Staubli VAL3: retrieveViews.pgx

public program retrieveViews(viewType& view_, num& idx_)
begin
  switch idx_
    case 0
      view_.path=IMM_IO_PTH
      view_.label="IMM"
      call views:appendNode(view_.nodes,"Safety")
      call views:appendNode(view_.nodes,"Machine")
      call views:appendNode(view_.nodes,"Ejectors")
      call views:appendNode(view_.nodes,"Cores")
      call views:appendNode(view_.nodes,"Mould")
      view_.type=view_.TYPE_TREEVIEW
    break
  endSwitch
end
